// TIA Portal project "Compressor" (V18)

(* hardware
DEVICE "S7-1200 station_1"  S7-1200 Station
   slot 0: "Rack_0"  S7-1200 Rack  Rack  V1.0
   slot 1: "PLC_1"  CPU 1212C DC/DC/Rly  6ES7 212-1HE40-0XB0  V4.6
   slot 2: "DQ 8xRelay_1"  SM 1222 DQ8 x relay  6ES7 222-1HF32-0XB0  V2.0
   slot 3: "AI 4xRTD_1"  6ES7 231-5PD30-0XB0  V1.0
*)

// ===== PLC "PLC_1"  CPU 1212C DC/DC/Rly =====

VAR_GLOBAL   // PLC tag table "Default tag table"
   "start" AT %I0.0 : Bool;
   "stop" AT %I0.1 : Bool;
   "motor1" AT %Q0.0 : Bool;
   "motor2" AT %Q0.1 : Bool;
   "motor3" AT %Q0.2 : Bool;
   "motor4" AT %Q0.3 : Bool;
   "tempError1" AT %Q0.4 : Bool;
   "tempError2" AT %Q0.5 : Bool;
   "tempError3" AT %Q1.0 : Bool;
   "tempError4" AT %Q1.1 : Bool;
   "pressureError" AT %Q1.2 : Bool;
   "sensor1" AT %IW64 : Word;
   "sensor2" AT %IW66 : Word;
   "sensor3" AT %IW68 : Word;
   "sensor4" AT %IW70 : Word;
   "pressureSensor" AT %IW72 : Word;
   "Tag_1" AT %MD0 : Real;
   "Tag_2" AT %MD3 : Real;
   "Tag_3" AT %MD4 : Real;
   "Tag_4" AT %MD8 : Real;
   "Tag_5" AT %MD12 : Real;
   "Tag_6" AT %MD16 : Real;
   "Tag_7" AT %MD20 : Real;
   "Tag_8" AT %M24.0 : Bool;
   "Tag_9" AT %M25.0 : Bool;
   "Tag_10" AT %M24.2 : Bool;
   "valve" AT %Q1.3 : Bool;
   "Tag_11" AT %M25.1 : Bool;
   "taeidOperator" AT %I0.2 : Bool;
   "Tag_12" AT %M26.1 : Bool;
   "Tag_13" AT %M26.2 : Bool;
   "Tag_14" AT %M27.1 : Bool;
END_VAR

ORGANIZATION_BLOCK "Main"   // OB1, LAD, ProgramCycle
TITLE = "Main Program Sweep (Cycle)"
{ S7_Optimized_Access := 'TRUE' }
VERSION : 0.1
   VAR_INPUT
      Initial_Call : Bool;   // Initial call of this OB
      Remanence : Bool;   // =True, if remanent data are available
   END_VAR
   VAR_TEMP   // added for the SCL form of the ladder/FBD networks
      _w1 : Bool;
      _w2 : Bool;
   END_VAR
BEGIN

REGION Network 1
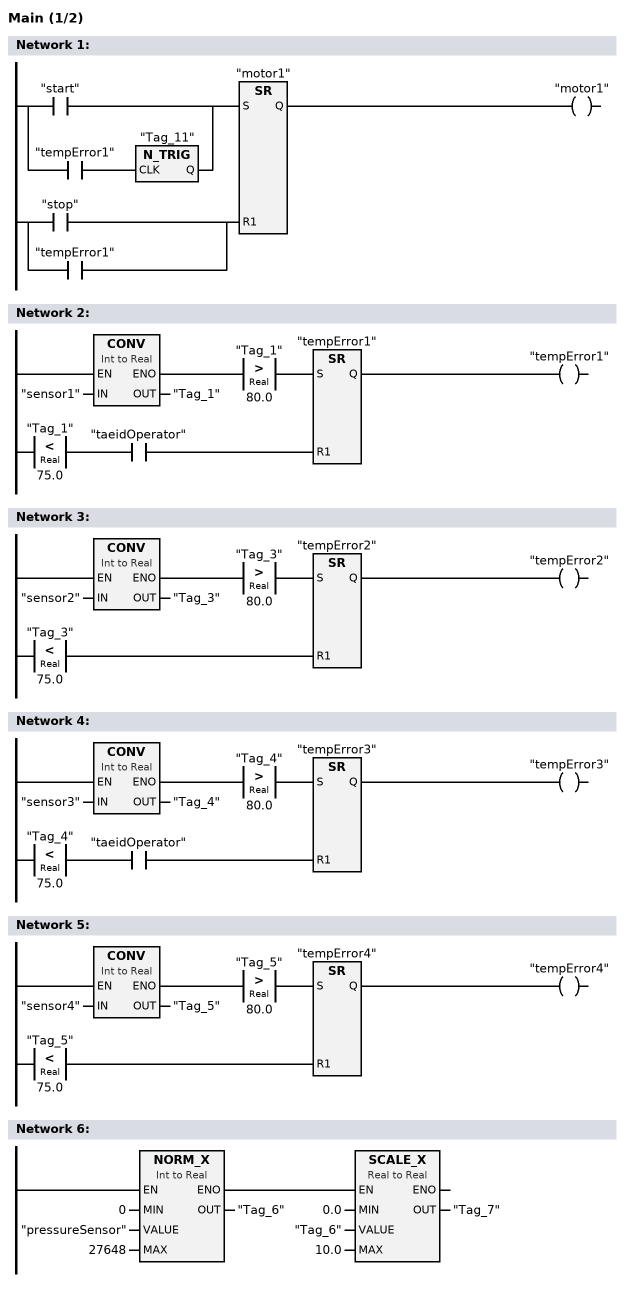
   RUNG wire#powerrail
      Contact( "start" )
      wire#w1
      S_SR(operand := "motor1", r1 := wire#w2)
      Coil( "motor1" )
   END_RUNG
   RUNG wire#powerrail
      Contact( "tempError1" )
      N_Trig( "Tag_11" )
   END_RUNG wire#w1
   RUNG wire#powerrail
      Contact( "stop" )
   END_RUNG wire#w2
   RUNG wire#powerrail
      Contact( "tempError1" )
   END_RUNG wire#w2
   // the same network as SCL:
   #_w1 := NOT "tempError1" AND "Tag_11";   // falling edge
   "Tag_11" := "tempError1";
   IF "start" OR #_w1 THEN
       "motor1" := TRUE;   // SR flip-flop
   END_IF;
   IF "stop" OR "tempError1" THEN "motor1" := FALSE; END_IF;
   "motor1" := "motor1";
END_REGION

REGION Network 2
   RUNG wire#powerrail
      { S7_Templates := "[SrcType := Int, DestType := Real]" } Convert(in := "sensor1", out => "Tag_1")
      { S7_Templates := "SrcType := Real" } GT_Contact(in1 := "Tag_1", in2 := 80.0)
      S_SR(operand := "tempError1", r1 := wire#w1)
      Coil( "tempError1" )
   END_RUNG
   RUNG wire#powerrail
      { S7_Templates := "SrcType := Real" } LT_Contact(in1 := "Tag_1", in2 := 75.0)
      Contact( "taeidOperator" )
   END_RUNG wire#w1
   // the same network as SCL:
   "Tag_1" := INT_TO_REAL("sensor1");
   IF "Tag_1" > 80.0 THEN
       "tempError1" := TRUE;   // SR flip-flop
   END_IF;
   IF ("Tag_1" < 75.0) AND "taeidOperator" THEN "tempError1" := FALSE; END_IF;
   "tempError1" := "tempError1";
END_REGION

REGION Network 3
   RUNG wire#powerrail
      { S7_Templates := "[SrcType := Int, DestType := Real]" } Convert(in := "sensor2", out => "Tag_3")
      { S7_Templates := "SrcType := Real" } GT_Contact(in1 := "Tag_3", in2 := 80.0)
      S_SR(operand := "tempError2", r1 := wire#w1)
      Coil( "tempError2" )
   END_RUNG
   RUNG wire#powerrail
      { S7_Templates := "SrcType := Real" } LT_Contact(in1 := "Tag_3", in2 := 75.0)
   END_RUNG wire#w1
   // the same network as SCL:
   "Tag_3" := INT_TO_REAL("sensor2");
   IF "Tag_3" > 80.0 THEN
       "tempError2" := TRUE;   // SR flip-flop
   END_IF;
   IF "Tag_3" < 75.0 THEN "tempError2" := FALSE; END_IF;
   "tempError2" := "tempError2";
END_REGION

REGION Network 4
   RUNG wire#powerrail
      { S7_Templates := "[SrcType := Int, DestType := Real]" } Convert(in := "sensor3", out => "Tag_4")
      { S7_Templates := "SrcType := Real" } GT_Contact(in1 := "Tag_4", in2 := 80.0)
      S_SR(operand := "tempError3", r1 := wire#w1)
      Coil( "tempError3" )
   END_RUNG
   RUNG wire#powerrail
      { S7_Templates := "SrcType := Real" } LT_Contact(in1 := "Tag_4", in2 := 75.0)
      Contact( "taeidOperator" )
   END_RUNG wire#w1
   // the same network as SCL:
   "Tag_4" := INT_TO_REAL("sensor3");
   IF "Tag_4" > 80.0 THEN
       "tempError3" := TRUE;   // SR flip-flop
   END_IF;
   IF ("Tag_4" < 75.0) AND "taeidOperator" THEN "tempError3" := FALSE; END_IF;
   "tempError3" := "tempError3";
END_REGION

REGION Network 5
   RUNG wire#powerrail
      { S7_Templates := "[SrcType := Int, DestType := Real]" } Convert(in := "sensor4", out => "Tag_5")
      { S7_Templates := "SrcType := Real" } GT_Contact(in1 := "Tag_5", in2 := 80.0)
      S_SR(operand := "tempError4", r1 := wire#w1)
      Coil( "tempError4" )
   END_RUNG
   RUNG wire#powerrail
      { S7_Templates := "SrcType := Real" } LT_Contact(in1 := "Tag_5", in2 := 75.0)
   END_RUNG wire#w1
   // the same network as SCL:
   "Tag_5" := INT_TO_REAL("sensor4");
   IF "Tag_5" > 80.0 THEN
       "tempError4" := TRUE;   // SR flip-flop
   END_IF;
   IF "Tag_5" < 75.0 THEN "tempError4" := FALSE; END_IF;
   "tempError4" := "tempError4";
END_REGION

REGION Network 6
   RUNG wire#powerrail
      { S7_Templates := "[SrcType := Int, DestType := Real]" } Normalize(min := 0, value := "pressureSensor", max := 27648, out => "Tag_6")
      { S7_Templates := "[SrcType := Real, DestType := Real]" } Scale(min := 0.0, value := "Tag_6", max := 10.0, out => "Tag_7")
   END_RUNG
   // the same network as SCL:
   "Tag_6" := NORM_X(MIN := 0, VALUE := "pressureSensor", MAX := 27648);
   "Tag_7" := SCALE_X(MIN := 0.0, VALUE := "Tag_6", MAX := 10.0);
END_REGION

REGION Network 7
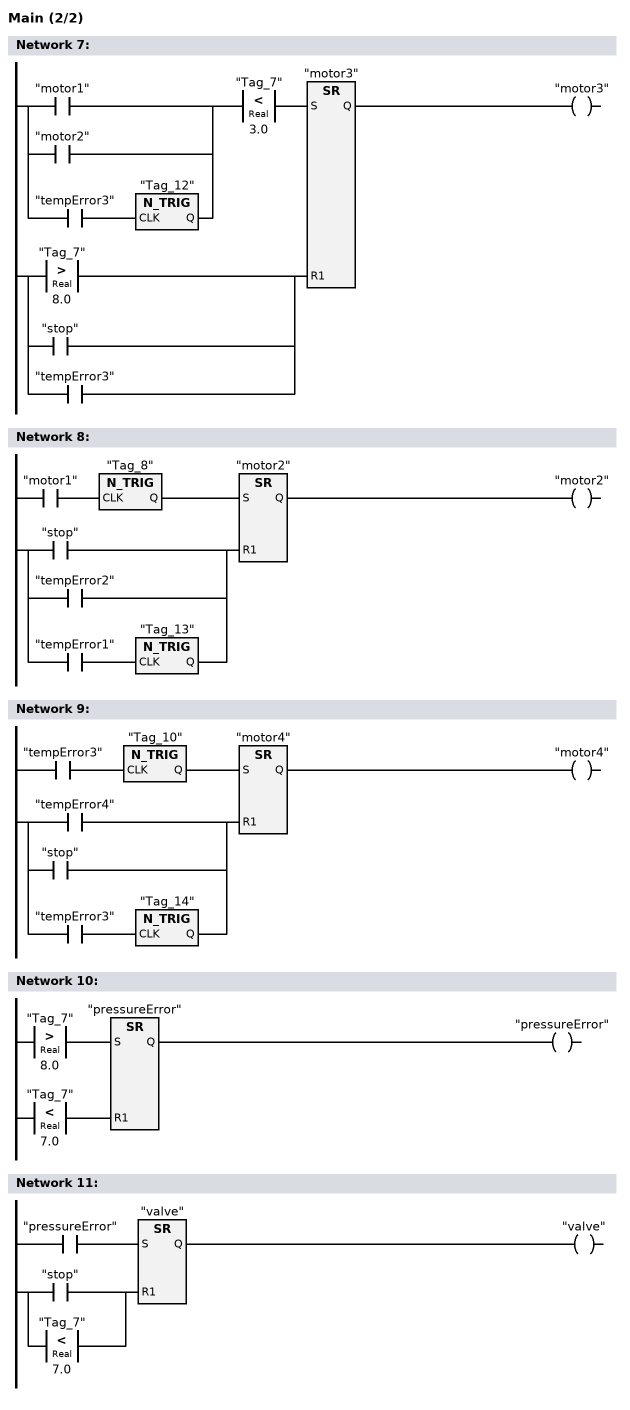
   RUNG wire#powerrail
      Contact( "motor1" )
      wire#w1
      { S7_Templates := "SrcType := Real" } LT_Contact(in1 := "Tag_7", in2 := 3.0)
      S_SR(operand := "motor3", r1 := wire#w2)
      Coil( "motor3" )
   END_RUNG
   RUNG wire#powerrail
      Contact( "motor2" )
   END_RUNG wire#w1
   RUNG wire#powerrail
      Contact( "tempError3" )
      N_Trig( "Tag_12" )
   END_RUNG wire#w1
   RUNG wire#powerrail
      { S7_Templates := "SrcType := Real" } GT_Contact(in1 := "Tag_7", in2 := 8.0)
   END_RUNG wire#w2
   RUNG wire#powerrail
      Contact( "stop" )
   END_RUNG wire#w2
   RUNG wire#powerrail
      Contact( "tempError3" )
   END_RUNG wire#w2
   // the same network as SCL:
   #_w1 := NOT "tempError3" AND "Tag_12";   // falling edge
   "Tag_12" := "tempError3";
   IF ("motor1" OR "motor2" OR #_w1) AND ("Tag_7" < 3.0) THEN
       "motor3" := TRUE;   // SR flip-flop
   END_IF;
   IF ("Tag_7" > 8.0) OR "stop" OR "tempError3" THEN "motor3" := FALSE; END_IF;
   "motor3" := "motor3";
END_REGION

REGION Network 8
   RUNG wire#powerrail
      Contact( "motor1" )
      N_Trig( "Tag_8" )
      S_SR(operand := "motor2", r1 := wire#w1)
      Coil( "motor2" )
   END_RUNG
   RUNG wire#powerrail
      Contact( "stop" )
   END_RUNG wire#w1
   RUNG wire#powerrail
      Contact( "tempError2" )
   END_RUNG wire#w1
   RUNG wire#powerrail
      Contact( "tempError1" )
      N_Trig( "Tag_13" )
   END_RUNG wire#w1
   // the same network as SCL:
   #_w1 := NOT "motor1" AND "Tag_8";   // falling edge
   "Tag_8" := "motor1";
   #_w2 := NOT "tempError1" AND "Tag_13";   // falling edge
   "Tag_13" := "tempError1";
   IF #_w1 THEN
       "motor2" := TRUE;   // SR flip-flop
   END_IF;
   IF "stop" OR "tempError2" OR #_w2 THEN "motor2" := FALSE; END_IF;
   "motor2" := "motor2";
END_REGION

REGION Network 9
   RUNG wire#powerrail
      Contact( "tempError3" )
      N_Trig( "Tag_10" )
      S_SR(operand := "motor4", r1 := wire#w1)
      Coil( "motor4" )
   END_RUNG
   RUNG wire#powerrail
      Contact( "tempError4" )
   END_RUNG wire#w1
   RUNG wire#powerrail
      Contact( "stop" )
   END_RUNG wire#w1
   RUNG wire#powerrail
      Contact( "tempError3" )
      N_Trig( "Tag_14" )
   END_RUNG wire#w1
   // the same network as SCL:
   #_w1 := NOT "tempError3" AND "Tag_10";   // falling edge
   "Tag_10" := "tempError3";
   #_w2 := NOT "tempError3" AND "Tag_14";   // falling edge
   "Tag_14" := "tempError3";
   IF #_w1 THEN
       "motor4" := TRUE;   // SR flip-flop
   END_IF;
   IF "tempError4" OR "stop" OR #_w2 THEN "motor4" := FALSE; END_IF;
   "motor4" := "motor4";
END_REGION

REGION Network 10
   RUNG wire#powerrail
      { S7_Templates := "SrcType := Real" } GT_Contact(in1 := "Tag_7", in2 := 8.0)
      S_SR(operand := "pressureError", r1 := wire#w1)
      Coil( "pressureError" )
   END_RUNG
   RUNG wire#powerrail
      { S7_Templates := "SrcType := Real" } LT_Contact(in1 := "Tag_7", in2 := 7.0)
   END_RUNG wire#w1
   // the same network as SCL:
   IF "Tag_7" > 8.0 THEN
       "pressureError" := TRUE;   // SR flip-flop
   END_IF;
   IF "Tag_7" < 7.0 THEN "pressureError" := FALSE; END_IF;
   "pressureError" := "pressureError";
END_REGION

REGION Network 11
   RUNG wire#powerrail
      Contact( "pressureError" )
      S_SR(operand := "valve", r1 := wire#w1)
      Coil( "valve" )
   END_RUNG
   RUNG wire#powerrail
      Contact( "stop" )
   END_RUNG wire#w1
   RUNG wire#powerrail
      { S7_Templates := "SrcType := Real" } LT_Contact(in1 := "Tag_7", in2 := 7.0)
   END_RUNG wire#w1
   // the same network as SCL:
   IF "pressureError" THEN
       "valve" := TRUE;   // SR flip-flop
   END_IF;
   IF "stop" OR ("Tag_7" < 7.0) THEN "valve" := FALSE; END_IF;
   "valve" := "valve";
END_REGION
END_ORGANIZATION_BLOCK